FUNCTION_BLOCK NormallyCloseSensor IMPLEMENTS I_Sensor
VAR
	input AT%I* : BOOL;
END_VAR

PROPERTY PUBLIC isActive : BOOL
GET
isActive	:=	NOT input;
END_GET
END_PROPERTY

PROPERTY PUBLIC isInactive : BOOL
GET
isInactive	:=	input;
END_GET
END_PROPERTY

END_FUNCTION_BLOCK

(* stored: Version 1.1.0.1, ProductVersion 3.1.4024.12
   POU NormallyCloseSensor: Id {27d68386-078b-4b0e-9b32-dae4341498a7}, SpecialFunc None
   Property isActive: Id {a6e23d46-d44d-4311-a84a-a94077605d34}
   Get Get: Id {78200d89-d84b-4ce4-ad38-d9bc5dbe3a7d}
   Property isInactive: Id {e5bb11c5-0b05-48eb-8819-d0266e029a89}
   Get Get: Id {e707d06b-35d1-4505-b6fb-ecccfa276ab9} *)
